TYPE typeHMIheader :
STRUCT
	
	stationstate: INT;
	homestate: INT; //home state for text list
	homestateColour: BOOL; //colour state of indicator

	anotherstate: BOOL;
	//faultstate: BOOL;
	//stationname: BOOL;
	flasher: BOOL;

	stationNameSelect: UINT; //station name selection
	cycleTypeFeedback: INT;
	
	isFaultState: BOOL; //colour change header
	FaultStateHeader: INT; //text change on header
	
	AnyStationFaultHeaderActive:BOOL;//colour change for global header
	AnyStationFaultHeader:INT; //text select for global header






END_STRUCT
END_TYPE

(* stored: Version 1.1.0.1, ProductVersion 3.1.4024.12
   DUT typeHMIheader: Id {c95c4980-1ece-470b-964a-d85f7da56a0f} *)
